TYPE ST_System_MachineParams :
STRUCT
	BMS									: ST_BMS_params;
	Interpowersupply					: ST_InternalPowerSupply_Params;
	Powerstack							: ST_Powerstack_Params;
	Coolingsystem						: ST_Coolingsystem_Params;
	NeutralTransformer					: ST_Neutraltransformer_Params;
	Protections							: ST_Protectionsystems_Params;
	Enclosure							: ST_Enclosure_Params;
	system								: ST_System_params;
	PNController						: ST_PNcontroller_params;
	IOT									: ST_IOT_params;
	Router								: ST_Router_params;
	PSB									: ST_peakshavebox_params;
END_STRUCT
END_TYPE

(* stored: Version 1.1.0.1, ProductVersion 3.1.4024.12
   DUT ST_System_MachineParams: Id {47922c1d-4635-4dcc-bc18-7c21b8f7cf41} *)
